PROGRAM POU_FBD
VAR
	input : BOOL;
	output : BOOL := false;
END_VAR

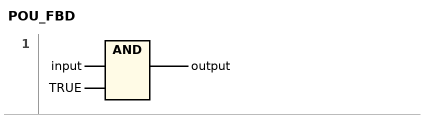
// NETWORK 1
output := input AND TRUE;

END_PROGRAM

(* stored: Version 1.1.0.1, ProductVersion 3.1.4024.12
   POU POU_FBD: Id {7412bda5-5393-4721-bd12-29c5bf7d46ed}, SpecialFunc None *)
